# B&R Automation Studio project 1st_testSTEPPER_SFL3
Automation Studio 4.9.2.46; technology packages: mappCockpit 5.12.0, mappMotion 5.12.2, mappSafety 5.12.2, mappView 5.12.1

## Configuration Config1

CPU 4PPC70.0702-20B, AutomationRuntime C4.90, Build 4.1.2, Safety 0.0, Vc V4.72.2

CPU 5PPC3100.KBU0-000, AutomationRuntime C4.90, Build 4.1.2, Safety 0.0, Vc V4.72.2

### Task classes (Cpu.sw)
```
Cyclic#4:
  Program <- Program.prg
NcDataObjects: CncProg <- CncProg.dob
Libraries: McBase, MpCnc, McAxGroup, MpBase, McPathGen, McAxis, McProgInt, McAcpAx, SfDomain, McStpAx, CoTrace, AsZip, FileIO, runtime
```

### Hardware
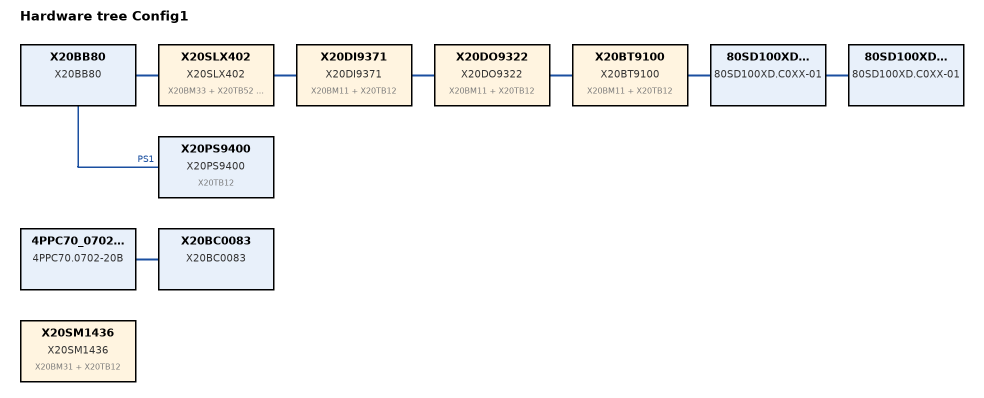
```
4PPC70_0702_20B : 4PPC70.0702-20B v1.5.2.0
  Connector IF2:
    ActivateDevice = 1
    Mode = Manual
    InternetAddress = 10.16.7.5
    SubnetMask = 255.255.0.0
    ActivateSnmp = 2
    DeviceParam = /EDDN=gei
  ConfigurationID = 1st_testSTEPPER_SFL3_Config1
  Cyclic1Duration = 2000
  Cyclic1Tolerance = 0
  ActivateOpcUa = 1
  OpcUaInformationModels_PV_Version = 1
  KeyMappingFile = VC\4PPC70_0702_20B.dis
80SD100XD.C0XX-01 : 80SD100XD.C0XX-01 v2.2.0.0  [X2X1 -> 80SD100XD.C0XX-01a.X2X2 [Cable Type=X2XCable, Length=10, Version=1.0.0.3]]
  Supervision = off
  FunctionModel/DriveConfiguration:
    ModuleParameters = StepperParameters
  FunctionModel/DriveConfiguration/ModuleParameters:
    McStepperTypeID = AcoposMicroConfig
    EncoderType = None
    ReferencePulse = yes
    RatedCurrent = 10.0
    MaximumCurrent = 15.0
    AxesNumber = 2
    FullStepThreshold = 1
    StallDetection = 0
    SmartCurrentControl = 0
    BrakeOutput = 1
    NumberOfDigitalInputs = 0
    NumberOfTriggers = 2
  FunctionModel/DriveConfiguration/Channel[1]/RealAxis:
    AxisReference = gAxisQZ
  FunctionModel/DriveConfiguration/Channel[1]/RealAxis/MechanicalElements/Gearbox:
    InputIsReadOnly = 0
    Input = 1
    OutputIsReadOnly = 0
    Output = 1
  FunctionModel/DriveConfiguration/Channel[1]/RealAxis/MechanicalElements/RotaryToLinearTransformation:
    ReferenceDistanceIsReadOnly = 0
    ReferenceDistance = 1
  FunctionModel/DriveConfiguration/Channel[1]/RealAxis/Motor:
    SteppingAngle = 1.8
  FunctionModel/DriveConfiguration/Channel[1]/RealAxis:
    EncoderLink = NoEncoder
  FunctionModel/DriveConfiguration/Channel[1]/RealAxis/Controller:
    ModeIsReadOnly = 0
    Mode = CurrentController
  FunctionModel/DriveConfiguration/Channel[1]/RealAxis/Controller/Mode/Current:
    StandstillCurrent = 0.20
    ConstantSpeedCurrent = 1.00
    SpeedChangeCurrent = 1.50
    FullStepThreshold = 0.0
    MotorSettlingTime = 1
    DelayedCurrentSwitchOff = 1
  FunctionModel/DriveConfiguration/Channel[1]/RealAxis/Homing:
    Mode = Direct
  FunctionModel/DriveConfiguration/Channel[1]/RealAxis/Homing/Mode:
    Position = 0.0
    ReferencePulse = NotUsed
  FunctionModel/DriveConfiguration/Channel[1]/RealAxis/Homing:
    RestorePositionVariable = 
  FunctionModel/DriveConfiguration/Channel[1]/RealAxis/StopReaction:
    DriveError = DecelerationLimit
  FunctionModel/DriveConfiguration/Channel[1]/RealAxis/MovementErrorLimits:
    PositionError = 1.0
  FunctionModel/DriveConfiguration/Channel[1]/RealAxis:
    JerkFilter = NotUsed
  FunctionModel/DriveConfiguration/Channel[1]/RealAxis/DigitalInputs/HomingSwitch:
    Source = NotUsed
    Level = High
  FunctionModel/DriveConfiguration/Channel[1]/RealAxis/DigitalInputs/PositiveLimitSwitch:
    Source = NotUsed
    Level = High
  FunctionModel/DriveConfiguration/Channel[1]/RealAxis/DigitalInputs/NegativeLimitSwitch:
    Source = NotUsed
    Level = High
  FunctionModel/DriveConfiguration/Channel[1]/RealAxis/DigitalInputs/Trigger1:
    Source = NotUsed
    Level = High
  FunctionModel/DriveConfiguration/Channel[1]/RealAxis/DigitalInputs/Trigger2:
    Source = NotUsed
    Level = High
  FunctionModel/DriveConfiguration/Channel[1]/RealAxis/DigitalInputs/Quickstop:
    Input = NotUsed
  FunctionModel/DriveConfiguration/Channel[1]/RealAxis/DigitalOutputs:
    BrakeControl = NotUsed
  FunctionModel/DriveConfiguration/Channel[2]/RealAxis:
    AxisReference = 
  FunctionModel/DriveConfiguration/Channel[2]/RealAxis/MechanicalElements/Gearbox:
    InputIsReadOnly = 0
    Input = 1
    OutputIsReadOnly = 0
    Output = 1
  FunctionModel/DriveConfiguration/Channel[2]/RealAxis/MechanicalElements/RotaryToLinearTransformation:
    ReferenceDistanceIsReadOnly = 0
    ReferenceDistance = 1
  FunctionModel/DriveConfiguration/Channel[2]/RealAxis/Motor:
    SteppingAngle = 1.8
  FunctionModel/DriveConfiguration/Channel[2]/RealAxis:
    EncoderLink = NoEncoder
  FunctionModel/DriveConfiguration/Channel[2]/RealAxis/Controller:
    ModeIsReadOnly = 0
    Mode = CurrentController
  FunctionModel/DriveConfiguration/Channel[2]/RealAxis/Controller/Mode/Current:
    StandstillCurrent = 0.3
    ConstantSpeedCurrent = 1.5
    SpeedChangeCurrent = 3
    FullStepThreshold = 0.0
    MotorSettlingTime = 1
    DelayedCurrentSwitchOff = 1
  FunctionModel/DriveConfiguration/Channel[2]/RealAxis/Homing:
    Mode = Direct
  FunctionModel/DriveConfiguration/Channel[2]/RealAxis/Homing/Mode:
    Position = 0.0
    ReferencePulse = NotUsed
  FunctionModel/DriveConfiguration/Channel[2]/RealAxis/Homing:
    RestorePositionVariable = 
  FunctionModel/DriveConfiguration/Channel[2]/RealAxis/StopReaction:
    DriveError = DecelerationLimit
  FunctionModel/DriveConfiguration/Channel[2]/RealAxis/MovementErrorLimits:
    PositionError = 1.0
  FunctionModel/DriveConfiguration/Channel[2]/RealAxis:
    JerkFilter = NotUsed
  FunctionModel/DriveConfiguration/Channel[2]/RealAxis/DigitalInputs/HomingSwitch:
    Source = NotUsed
    Level = High
  FunctionModel/DriveConfiguration/Channel[2]/RealAxis/DigitalInputs/PositiveLimitSwitch:
    Source = NotUsed
    Level = High
  FunctionModel/DriveConfiguration/Channel[2]/RealAxis/DigitalInputs/NegativeLimitSwitch:
    Source = NotUsed
    Level = High
  FunctionModel/DriveConfiguration/Channel[2]/RealAxis/DigitalInputs/Trigger1:
    Source = NotUsed
    Level = High
  FunctionModel/DriveConfiguration/Channel[2]/RealAxis/DigitalInputs/Trigger2:
    Source = NotUsed
    Level = High
  FunctionModel/DriveConfiguration/Channel[2]/RealAxis/DigitalInputs/Quickstop:
    Input = NotUsed
  FunctionModel/DriveConfiguration/Channel[2]/RealAxis/DigitalOutputs:
    BrakeControl = NotUsed
80SD100XD.C0XX-01a : 80SD100XD.C0XX-01 v2.2.0.0  [X2X1 -> X20BT9100.X2X1 [Cable Type=X2XCable, Length=10, Version=1.0.0.3]]
  Supervision = off
  FunctionModel/DriveConfiguration:
    ModuleParameters = StepperParameters
  FunctionModel/DriveConfiguration/ModuleParameters:
    McStepperTypeID = AcoposMicroConfig
    EncoderType = None
    ReferencePulse = yes
    RatedCurrent = 10.0
    MaximumCurrent = 15.0
    AxesNumber = 2
    FullStepThreshold = 1
    StallDetection = 0
    SmartCurrentControl = 0
    BrakeOutput = 1
    NumberOfDigitalInputs = 0
    NumberOfTriggers = 2
  FunctionModel/DriveConfiguration/Channel[1]/RealAxis:
    AxisReference = gAxisQX
  FunctionModel/DriveConfiguration/Channel[1]/RealAxis/MechanicalElements/Gearbox:
    InputIsReadOnly = 0
    Input = 1
    OutputIsReadOnly = 0
    Output = 1
  FunctionModel/DriveConfiguration/Channel[1]/RealAxis/MechanicalElements/RotaryToLinearTransformation:
    ReferenceDistanceIsReadOnly = 0
    ReferenceDistance = 1
  FunctionModel/DriveConfiguration/Channel[1]/RealAxis/Motor:
    SteppingAngle = 1.8
  FunctionModel/DriveConfiguration/Channel[1]/RealAxis:
    EncoderLink = NoEncoder
  FunctionModel/DriveConfiguration/Channel[1]/RealAxis/Controller:
    ModeIsReadOnly = 0
    Mode = CurrentController
  FunctionModel/DriveConfiguration/Channel[1]/RealAxis/Controller/Mode/Current:
    StandstillCurrent = 0.20
    ConstantSpeedCurrent = 1.00
    SpeedChangeCurrent = 1.50
    FullStepThreshold = 0.0
    MotorSettlingTime = 1
    DelayedCurrentSwitchOff = 1
  FunctionModel/DriveConfiguration/Channel[1]/RealAxis/Homing:
    Mode = Direct
  FunctionModel/DriveConfiguration/Channel[1]/RealAxis/Homing/Mode:
    Position = 0.0
    ReferencePulse = NotUsed
  FunctionModel/DriveConfiguration/Channel[1]/RealAxis/Homing:
    RestorePositionVariable = 
  FunctionModel/DriveConfiguration/Channel[1]/RealAxis/StopReaction:
    DriveError = DecelerationLimit
  FunctionModel/DriveConfiguration/Channel[1]/RealAxis/MovementErrorLimits:
    PositionError = 1.0
  FunctionModel/DriveConfiguration/Channel[1]/RealAxis:
    JerkFilter = NotUsed
  FunctionModel/DriveConfiguration/Channel[1]/RealAxis/DigitalInputs/HomingSwitch:
    Source = NotUsed
    Level = High
  FunctionModel/DriveConfiguration/Channel[1]/RealAxis/DigitalInputs/PositiveLimitSwitch:
    Source = NotUsed
    Level = High
  FunctionModel/DriveConfiguration/Channel[1]/RealAxis/DigitalInputs/NegativeLimitSwitch:
    Source = NotUsed
    Level = High
  FunctionModel/DriveConfiguration/Channel[1]/RealAxis/DigitalInputs/Trigger1:
    Source = NotUsed
    Level = High
  FunctionModel/DriveConfiguration/Channel[1]/RealAxis/DigitalInputs/Trigger2:
    Source = NotUsed
    Level = High
  FunctionModel/DriveConfiguration/Channel[1]/RealAxis/DigitalInputs/Quickstop:
    Input = NotUsed
  FunctionModel/DriveConfiguration/Channel[1]/RealAxis/DigitalOutputs:
    BrakeControl = NotUsed
  FunctionModel/DriveConfiguration/Channel[2]/RealAxis:
    AxisReference = gAxisQY
  FunctionModel/DriveConfiguration/Channel[2]/RealAxis/MechanicalElements/Gearbox:
    InputIsReadOnly = 0
    Input = 1
    OutputIsReadOnly = 0
    Output = 1
  FunctionModel/DriveConfiguration/Channel[2]/RealAxis/MechanicalElements/RotaryToLinearTransformation:
    ReferenceDistanceIsReadOnly = 0
    ReferenceDistance = 1
  FunctionModel/DriveConfiguration/Channel[2]/RealAxis/Motor:
    SteppingAngle = 1.8
  FunctionModel/DriveConfiguration/Channel[2]/RealAxis:
    EncoderLink = NoEncoder
  FunctionModel/DriveConfiguration/Channel[2]/RealAxis/Controller:
    ModeIsReadOnly = 0
    Mode = CurrentController
  FunctionModel/DriveConfiguration/Channel[2]/RealAxis/Controller/Mode/Current:
    StandstillCurrent = 0.20
    ConstantSpeedCurrent = 1.00
    SpeedChangeCurrent = 1.50
    FullStepThreshold = 0.0
    MotorSettlingTime = 1
    DelayedCurrentSwitchOff = 1
  FunctionModel/DriveConfiguration/Channel[2]/RealAxis/Homing:
    Mode = Direct
  FunctionModel/DriveConfiguration/Channel[2]/RealAxis/Homing/Mode:
    Position = 0.0
    ReferencePulse = NotUsed
  FunctionModel/DriveConfiguration/Channel[2]/RealAxis/Homing:
    RestorePositionVariable = 
  FunctionModel/DriveConfiguration/Channel[2]/RealAxis/StopReaction:
    DriveError = DecelerationLimit
  FunctionModel/DriveConfiguration/Channel[2]/RealAxis/MovementErrorLimits:
    PositionError = 1.0
  FunctionModel/DriveConfiguration/Channel[2]/RealAxis:
    JerkFilter = NotUsed
  FunctionModel/DriveConfiguration/Channel[2]/RealAxis/DigitalInputs/HomingSwitch:
    Source = NotUsed
    Level = High
  FunctionModel/DriveConfiguration/Channel[2]/RealAxis/DigitalInputs/PositiveLimitSwitch:
    Source = NotUsed
    Level = High
  FunctionModel/DriveConfiguration/Channel[2]/RealAxis/DigitalInputs/NegativeLimitSwitch:
    Source = NotUsed
    Level = High
  FunctionModel/DriveConfiguration/Channel[2]/RealAxis/DigitalInputs/Trigger1:
    Source = NotUsed
    Level = High
  FunctionModel/DriveConfiguration/Channel[2]/RealAxis/DigitalInputs/Trigger2:
    Source = NotUsed
    Level = High
  FunctionModel/DriveConfiguration/Channel[2]/RealAxis/DigitalInputs/Quickstop:
    Input = NotUsed
  FunctionModel/DriveConfiguration/Channel[2]/RealAxis/DigitalOutputs:
    BrakeControl = NotUsed
X20BB80 : X20BB80 v1.0.2.0
X20BC0083 : X20BC0083 v2.11.1.0  [PLK2 -> 4PPC70_0702_20B.IF1 (NodeNumber=1) [Cable Type=PowerlinkCable, Length=10, Version=1.0.0.3]; SL -> X20BB80.SL1]
  Supervision = off
X20BM11 : X20BM11 v1.0.0.1  [X2X1 -> X20BM33.X2X2]
X20BM11a : X20BM11 v1.0.0.1  [X2X1 -> X20BM11.X2X2]
X20BM11b : X20BM11 v1.0.0.1  [X2X1 -> X20BM11a.X2X2]
X20BM31 : X20BM31 v1.0.0.1
X20BM33 : X20BM33 v1.0.0.6  [X2X1 -> X20BB80.IF1]
X20BT9100 : X20BT9100 v1.1.0.0  [SS1 -> X20TB12d.SS; SL -> X20BM11b.SL1]
  Supervision = off
X20DI9371 : X20DI9371 v1.1.0.0  [SS1 -> X20TB12b.SS; SL -> X20BM11.SL1]
  Supervision = off
X20DO9322 : X20DO9322 v1.3.0.0  [SS1 -> X20TB12c.SS; SL -> X20BM11a.SL1]
  Supervision = off
X20PS9400 : X20PS9400 v1.4.0.0  [SS1 -> X20TB12a.SS; PS -> X20BB80.PS1]
  Supervision = off
X20SLX402 : X20SLX402 v2.2.0.0  [SS1 -> X20TB52.SS; SS2 -> X20TB52a.SS; SL -> X20BM33.SL1]
  Supervision = off
  DigitalOutput01 = viaSafeLOGIC
  DigitalOutput02 = viaSafeLOGIC
X20SM1436 : X20SM1436 v2.2.0.0  [SS1 -> X20TB12.SS; SL -> X20BM31.SL1]
  FunctionModel/DriveConfiguration:
    ModuleParameters = StepperParameters
  FunctionModel/DriveConfiguration/ModuleParameters:
    McStepperTypeID = X20Config
    EncoderType = Incremental
    ReferencePulse = yes
    RatedCurrent = 3.0
    MaximumCurrent = 3.51
    AxesNumber = 1
    FullStepThreshold = 1
    StallDetection = 1
    SmartCurrentControl = 0
    BrakeOutput = 0
    NumberOfDigitalInputs = 3
    NumberOfTriggers = 1
  FunctionModel/DriveConfiguration/Channel[1]/RealAxis:
    AxisReference = 
  FunctionModel/DriveConfiguration/Channel[1]/RealAxis/MechanicalElements/Gearbox:
    InputIsReadOnly = 0
    Input = 1
    OutputIsReadOnly = 0
    Output = 1
  FunctionModel/DriveConfiguration/Channel[1]/RealAxis/MechanicalElements/RotaryToLinearTransformation:
    ReferenceDistanceIsReadOnly = 0
    ReferenceDistance = 1
  FunctionModel/DriveConfiguration/Channel[1]/RealAxis/Motor:
    SteppingAngle = 1.8
  FunctionModel/DriveConfiguration/Channel[1]/RealAxis:
    EncoderLink = NoEncoder
  FunctionModel/DriveConfiguration/Channel[1]/RealAxis/Controller:
    ModeIsReadOnly = 0
    Mode = CurrentController
  FunctionModel/DriveConfiguration/Channel[1]/RealAxis/Controller/Mode/Current:
    StandstillCurrent = 0.09
    ConstantSpeedCurrent = 0.45
    SpeedChangeCurrent = 0.9
    FullStepThreshold = 0.0
    MotorSettlingTime = 1
    DelayedCurrentSwitchOff = 1
  FunctionModel/DriveConfiguration/Channel[1]/RealAxis/Homing:
    Mode = Direct
  FunctionModel/DriveConfiguration/Channel[1]/RealAxis/Homing/Mode:
    Position = 0.0
    ReferencePulse = NotUsed
  FunctionModel/DriveConfiguration/Channel[1]/RealAxis/Homing:
    RestorePositionVariable = 
  FunctionModel/DriveConfiguration/Channel[1]/RealAxis/StopReaction:
    DriveError = DecelerationLimit
  FunctionModel/DriveConfiguration/Channel[1]/RealAxis/MovementErrorLimits:
    PositionError = 1.0
    StallDetectionConfiguration = NotUsed
  FunctionModel/DriveConfiguration/Channel[1]/RealAxis:
    JerkFilter = NotUsed
  FunctionModel/DriveConfiguration/Channel[1]/RealAxis/DigitalInputs/HomingSwitch:
    Source = NotUsed
    Level = High
  FunctionModel/DriveConfiguration/Channel[1]/RealAxis/DigitalInputs/PositiveLimitSwitch:
    Source = NotUsed
    Level = High
  FunctionModel/DriveConfiguration/Channel[1]/RealAxis/DigitalInputs/NegativeLimitSwitch:
    Source = NotUsed
    Level = High
  FunctionModel/DriveConfiguration/Channel[1]/RealAxis/DigitalInputs/Trigger1:
    Source = NotUsed
    Level = High
  FunctionModel/DriveConfiguration/Channel[1]/RealAxis/DigitalInputs/Trigger2:
    Source = NotUsed
    Level = High
  FunctionModel/DriveConfiguration/Channel[1]/RealAxis/DigitalInputs/Quickstop:
    Input = NotUsed
  FunctionModel/DriveConfiguration/Channel[1]/RealAxis/DigitalOutputs:
    BrakeControl = NotUsed
X20TB12 : X20TB12 v1.0.0.0
X20TB12a : X20TB12 v1.0.0.0
X20TB12b : X20TB12 v1.0.0.0
X20TB12c : X20TB12 v1.0.0.0
X20TB12d : X20TB12 v1.0.0.0
X20TB52 : X20TB52 v1.0.0.2
X20TB52a : X20TB52 v1.0.0.2
```

### Config_1.axesgroup - 4PPC70_0702_20B/mappMotion/3AxesCNCXYZ/Config_1.axesgroup
```
Element gCncXYZ (Type=axesgroup)
  Type = PathGenAxesGroup
    ProcessingTaskClass = 1
    License = 1
    PhysicalAxes:
      JointAxes:
        JointAxis[1]:
          Name = QX
          AxisRef = gAxisQX
        JointAxis[2]:
          Name = QY
          AxisRef = gAxisQY
        JointAxis[3]:
          Name = QZ
          AxisRef = gAxisQZ
    MechanicalSystem:
      MechSysRef = MechSys_3AxCNCXYZ
    BasicSettings:
      ModalDataBehaviour = ResetToDefault
      GeometryPlanning:
        RoundingMode = Standard
        MaxCornerDeviation = 0.0
        MaxTangentialTransitionDeviation = 0.0
        MaxRadiusDeviation = 0.001
        WorkingPlane = XY
      TrajectoryPlanning = Basic
        LimitCheckResolution = UserDefinedTime
          Time = 0.01
        BufferTime = UserDefinedTime
          Time = 0.1
    AxesGroupFeatures:
      FeatureRef[1] = Feature_Programs
      FeatureRef[2] = Feature_Jogging
  Alarms = None
```

### Config_3.mechanicalsystem - 4PPC70_0702_20B/mappMotion/3AxesCNCXYZ/Config_3.mechanicalsystem
```
Element MechSys_3AxCNCXYZ (Type=mechanicalsystem)
  Type = 3AxesCNC
    Subtype = 3AxesCNCXYZ
      CoordinatesNames = Default
        XCoordinateName = X
        YCoordinateName = Y
        ZCoordinateName = Z
      WireFrameModel = Standard
        FlangeToTcp = ConnectionLine
          Distance = 0.0
      JointAxesPositionLimits:
        JointAxis[1] = UseAxisLimits
        JointAxis[2] = UseAxisLimits
        JointAxis[3] = UseAxisLimits
```

- Safety project (password-protected, skipped)

### Config_2.axis - 5PPC3100_KBU2_000/mappMotion/3AxesCNCXYZ/Config_2.axis
```
Element gAxisQX (Type=axis)
  BaseTypeIsReadOnly = 0
  BaseType = RotaryPeriodic
    MeasurementUnitIsReadOnly = 0
    MeasurementUnit = 17476
    MeasurementResolutionIsReadOnly = 0
    MeasurementResolution = 0.01
    CountDirectionIsReadOnly = 0
    CountDirection = Standard
    PeriodSettings:
      Period = 360.0
  MovementLimitsIsReadOnly = 0
  MovementLimits = Internal
    Position:
      LowerLimitMin = -1.79769313486231E308
      UpperLimitMax = 1.79769313486231E308
      LowerLimit = -1000.0
      UpperLimit = 1000.0
    VelocityIsReadOnly = 0
    Velocity:
      VelocityMax = 3.4E38
      Velocity = 200
    AccelerationIsReadOnly = 0
    Acceleration:
      AccelerationMax = 3.4E38
      Acceleration = 50.0
    DecelerationIsReadOnly = 0
    Deceleration:
      DecelerationMax = 3.4E38
      Deceleration = 50.0
  Alarms = None
Element gAxisQY (Type=axis)
  BaseTypeIsReadOnly = 0
  BaseType = RotaryPeriodic
    MeasurementUnitIsReadOnly = 0
    MeasurementUnit = 17476
    MeasurementResolutionIsReadOnly = 0
    MeasurementResolution = 0.01
    CountDirectionIsReadOnly = 0
    CountDirection = Standard
    PeriodSettings:
      Period = 360.0
  MovementLimitsIsReadOnly = 0
  MovementLimits = Internal
    Position:
      LowerLimitMin = -1.79769313486231E308
      UpperLimitMax = 1.79769313486231E308
      LowerLimit = -1000.0
      UpperLimit = 1000.0
    VelocityIsReadOnly = 0
    Velocity:
      VelocityMax = 3.4E38
      Velocity = 200
    AccelerationIsReadOnly = 0
    Acceleration:
      AccelerationMax = 3.4E38
      Acceleration = 50.0
    DecelerationIsReadOnly = 0
    Deceleration:
      DecelerationMax = 3.4E38
      Deceleration = 50.0
  Alarms = None
Element gAxisQZ (Type=axis)
  BaseTypeIsReadOnly = 0
  BaseType = LinearBounded
    MeasurementUnit = 5066068
    MeasurementResolutionIsReadOnly = 0
    MeasurementResolution = 0.01
    CountDirectionIsReadOnly = 0
    CountDirection = Standard
  MovementLimitsIsReadOnly = 0
  MovementLimits = Internal
    Position:
      LowerLimitMin = -1.79769313486231E308
      UpperLimitMax = 1.79769313486231E308
      LowerLimit = -1000.0
      UpperLimit = 1000.0
    VelocityIsReadOnly = 0
    Velocity:
      VelocityMax = 3.4E38
      Velocity = 200
    AccelerationIsReadOnly = 0
    Acceleration:
      AccelerationMax = 3.4E38
      Acceleration = 50.0
    DecelerationIsReadOnly = 0
    Deceleration:
      DecelerationMax = 3.4E38
      Deceleration = 50.0
  Alarms = None
```

## Logical view

Binary libraries used (declarations not repeated): operator, runtime, astime, AsIecCon, McBase, MpCnc 5.12.2, McAxGroup 5.12.2, MpBase, McPathGen 5.12.2, McAxis, McProgInt 5.12.2, McAcpAx 5.12.2, SfDomain, McStpAx 5.12.2, CoTrace 5.12.0, AsZip, FileIO


### Data object Logical/CncProg (Cnc)

#### CncProg.cnc - CNC program (G-Code)
```
%001 (CncProgram)

N10 G90 (coordonnées absolues)
N20 F300  (vitesse de rotation en U/min)

N30 G04 2   (temps d'attente de 2s)

N50 G01 X50 Y50 Z50   (mouvement linéaire)

N60 G04 2    (temps d'attente de 2s)

N100 G01 X0 Y0 Z0  (retour vers O)

N999 M30
```

### Program Logical/Program (IEC)

#### Variables.var
```iecst
VAR
	MpCnc3axis_0 : MpCnc3Axis;
	CncParameters : MpCnc3AxisParType;
END_VAR
```

#### Main.st
```iecst
PROGRAM _INIT

	MpCnc3axis_0.MpLink := ADR(gCncXYZ);
	MpCnc3axis_0.Enable := TRUE;
	MpCnc3axis_0.Parameters := ADR(CncParameters);

	MpCnc3axis_0.Override := 100.0;
	CncParameters.ProgramName := 'CncProg';

END_PROGRAM

PROGRAM _CYCLIC

	MpCnc3axis_0();

END_PROGRAM

PROGRAM _EXIT

	MpCnc3axis_0.Enable := FALSE;
	MpCnc3axis_0.Power  := FALSE;
	MpCnc3axis_0.Home   := FALSE;
	MpCnc3axis_0();

END_PROGRAM
```

Listed in the project but not available here: Logical/Global.typ, Logical/Global.var
